RoboDK station: Example-01.b-Robot Drilling - KUKA.rdk

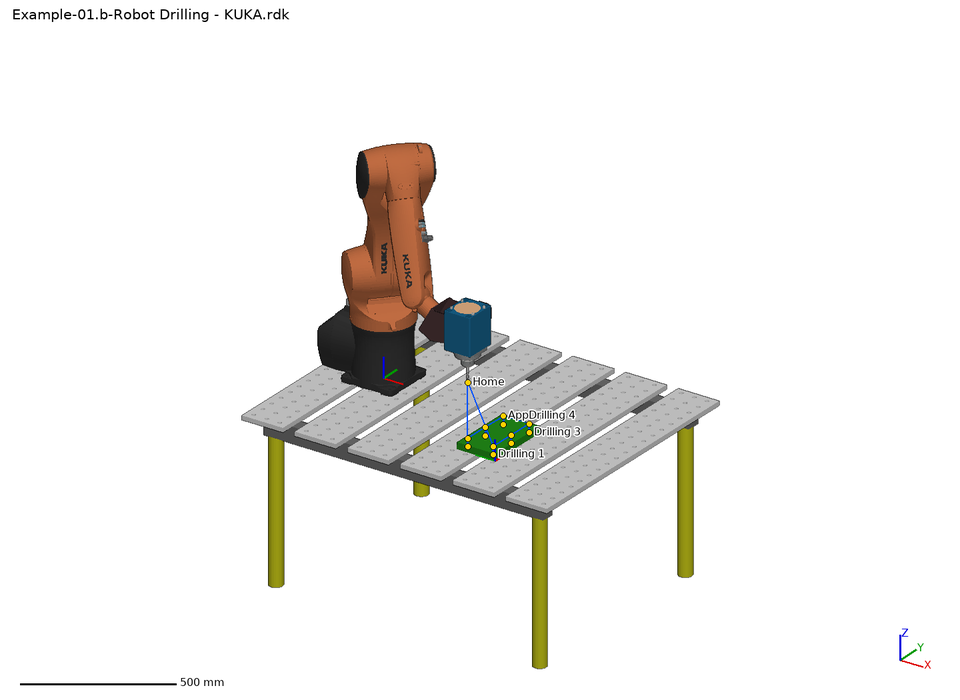
[picture v0: the station drawn from its stored meshes, robots at their saved joint values, targets as dots, program paths as lines]
Station Example-01.b-Robot Drilling - KUKA (saved by RoboDK 5.2.3). Poses are relative to the parent item; angles as X-Y-Z fixed-axis rotations.
  - frame KUKA KR 10 R900 sixx Base at (0, 0, 0) mm
    - robot KUKA KR 10 R900 sixx: 6 axes, payload 10 kg, reach 901 mm, repeatability 0.03 mm, weight 52 kg
        modified DH rows (alpha deg, a mm, theta deg, d mm): 0, 0, 0, 400; -90, 25, 0, 0; 0, 455, -90, 0; -90, 35, 0, 420; 90, 0, 0, 0; -90, 0, 180, 80
        joint limits [-170, -190, -120, -185, -120, -350] to [170, 45, 156, 185, 120, 350]; home [0, -90, 90, 0, 0, 0]; saved at [40.166, -71.395, 131.333, 60.015, -40.159, -30.067]
      - tool Spindle, TCP at (116.06, 0, 219.48) mm, rotated rx 0 ry 60 rz 0 deg, size 260.9 x 152 x 222 mm, geometry from Little spindle.step
    - object Table at (380, 0, 0) mm, size 1193.8 x 965.2 x 609.6 mm, geometry from welding_table.sld
  - frame Part 1 at (640.29, -290, 0) mm, rotated rx 0 ry 0 rz 90 deg
    - object Drilling at (0, 0, 0) mm, size 250 x 150 x 25 mm, geometry from Drilling.step
    - target Home (Cartesian target) at (25, 125, 235) mm, rotated rx -180 ry 0 rz 90 deg; joints [40.166, -71.395, 131.333, 60.015, -40.159, -30.067] of KUKA KR 10 R900 sixx
    - target Drilling 1 (Cartesian target) at (25, 25, 5) mm, rotated rx -180 ry 0 rz 90 deg; joints [9.438, -40.7, 124.04, 9.501, -83.43, -1.097] of KUKA KR 10 R900 sixx
    - target Drilling 2 (Cartesian target) at (125, 25, 5) mm, rotated rx -180 ry 0 rz 90 deg; joints [-57.379, -35.838, 153.204, -126.861, -32.652, -27.341] of KUKA KR 10 R900 sixx
    - target Drilling 3 (Cartesian target) at (225, 25, 5) mm, rotated rx -180 ry 0 rz 90 deg; joints [-40.958, -39.896, 145.068, -120.051, -44.318, -16.433] of KUKA KR 10 R900 sixx
    - target Drilling 4 (Cartesian target) at (225, 125, 5) mm, rotated rx -180 ry 0 rz 90 deg; joints [-52.695, -41.042, 135.387, -140.548, -49.797, -3.447] of KUKA KR 10 R900 sixx
    - target Drilling 5 (Cartesian target) at (125, 125, 5) mm, rotated rx -180 ry 0 rz 90 deg; joints [-67.057, -40.548, 142.134, -152.596, -42.703, -6.629] of KUKA KR 10 R900 sixx
    - target Drilling 6 (Cartesian target) at (25, 125, 5) mm, rotated rx -180 ry 0 rz 90 deg; joints [-85.161, -39.839, 145.27, 6.321, 37.844, 177.903] of KUKA KR 10 R900 sixx
    - target AppDrilling 1 (Cartesian target) at (25, 25, 35) mm, rotated rx -180 ry 0 rz 90 deg; joints [9.438, -44.943, 125.087, 9.577, -80.279, -1.632] of KUKA KR 10 R900 sixx
    - target AppDrilling 2 (Cartesian target) at (125, 25, 35) mm, rotated rx -180 ry 0 rz 90 deg; joints [-57.379, -42.811, 155.1, -132.596, -35.902, -20.405] of KUKA KR 10 R900 sixx
    - target AppDrilling 3 (Cartesian target) at (225, 25, 35) mm, rotated rx -180 ry 0 rz 90 deg; joints [-40.958, -45.85, 146.604, -123.74, -46.654, -11.173] of KUKA KR 10 R900 sixx
    - target AppDrilling 4 (Cartesian target) at (225, 125, 35) mm, rotated rx -180 ry 0 rz 90 deg; joints [-52.695, -46.066, 136.671, -142.417, -52.723, -0.461] of KUKA KR 10 R900 sixx
    - target AppDrilling 5 (Cartesian target) at (125, 125, 35) mm, rotated rx -180 ry 0 rz 90 deg; joints [-67.057, -46.187, 143.58, -154.493, -46.459, -3.968] of KUKA KR 10 R900 sixx
    - target AppDrilling 6 (Cartesian target) at (25, 125, 35) mm, rotated rx -180 ry 0 rz 90 deg; joints [-85.161, -45.815, 146.813, 5.766, 42.253, 178.629] of KUKA KR 10 R900 sixx
  - program DrillingPart (22 instructions, listed below)
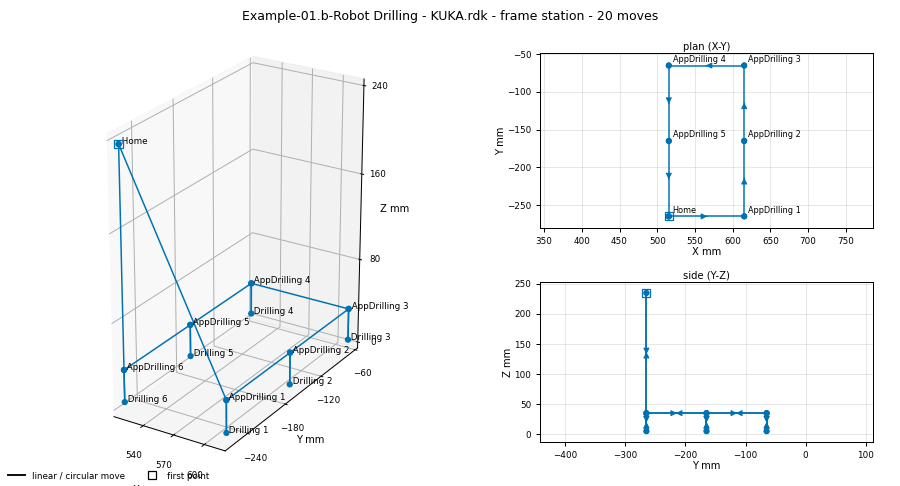
[picture p0: tool path of Example-01.b-Robot Drilling - KUKA.rdk in frame station, 20 of 20 moves have a stored position in this frame; points joined in program order, loops and branches not executed]

--- program DrillingPart (robot KUKA KR 10 R900 sixx) ---
  Set Ref.: Part 1
  Set Tool: Spindle
  MoveJ (Home)
  MoveL (AppDrilling 1)
  MoveL (Drilling 1)
  MoveL (AppDrilling 1)
  MoveL (AppDrilling 2)
  MoveL (Drilling 2)
  MoveL (AppDrilling 2)
  MoveL (AppDrilling 3)
  MoveL (Drilling 3)
  MoveL (AppDrilling 3)
  MoveL (AppDrilling 4)
  MoveL (Drilling 4)
  MoveL (AppDrilling 4)
  MoveL (AppDrilling 5)
  MoveL (Drilling 5)
  MoveL (AppDrilling 5)
  MoveL (AppDrilling 6)
  MoveL (Drilling 6)
  MoveL (AppDrilling 6)
  MoveL (Home)
